Fanuc KAREL source: kc00014.KL

-- PROVISIONAL review KL for V940-1; original PC SHA256 b16187b9065a407b52f5612114f007d651519774003d3ad67d80dee351bc12c6
-- Incomplete behavior may be omitted. Consult companion uncertainty JSON. Do not deploy.
PROGRAM KC00014
%NOLOCKGROUP
BEGIN
  -- V9_ZERO_TABLE_METADATA_HINT layout=0002_ascii; no indexed target words; source/name/runtime held
  -- UNRESOLVED_PC offsets 5-15; opcodes 27,31,23
  -- UNRESOLVED_PC offsets 20-24; opcodes 7F
END KC00014
